{attribute 'qualified_only'}
VAR_GLOBAL
	
	// A string to test reading.
	sReadTest : STRING := 'The quick brown fox jumps over the lazy dog.';
	
END_VAR

(* stored: Version 1.1.0.1, ProductVersion 3.1.4024.12
   GVL GK: Id {b6a38a92-5945-487d-9937-d60b9f91761f} *)
